% RSLogix 500 project PROJECT10.RSS, saved by version 8.30.00.16 %
PROJECT "PROJ_9"    % processor: Bul.1763 MicroLogix 1100 Series B %

PROGRAM FILES
  LAD 2 "MAIN"  5 rungs
  LAD 3 "I/O"  11 rungs
  LAD 4 "CONTROL"  6 rungs
  LAD 5 "ALARMS"  5 rungs

DATA FILES
  O0 OUTPUT  5 elements
  I1 INPUT  7 elements
  S2 STATUS  66 elements
  B3 BINARY  2 elements
  T4 TIMER  4 elements
  C5 COUNTER  1 elements
  R6 CONTROL  1 elements
  N7 INTEGER  2 elements
  F8 FLOAT  1 elements

LADDER 2 "MAIN"
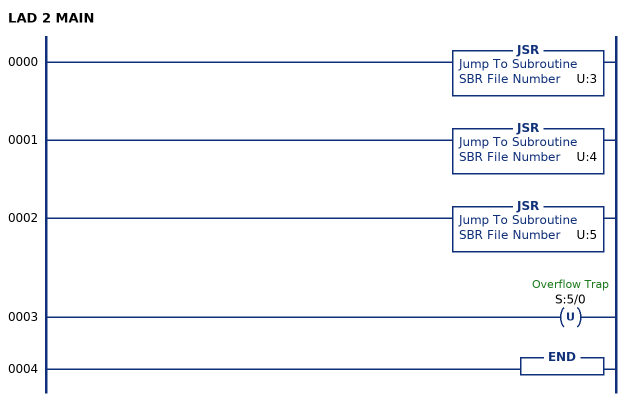
% Rung: 0 %
SOR JSR U:3 EOR
% Rung: 1 %
SOR JSR U:4 EOR
% Rung: 2 %
SOR JSR U:5 EOR
% Rung: 3 %
SOR OTU S:5/0 EOR
%   S:5/0  "Overflow Trap" %
% Rung: 4 %
SOR END EOR

LADDER 3 "I/O"
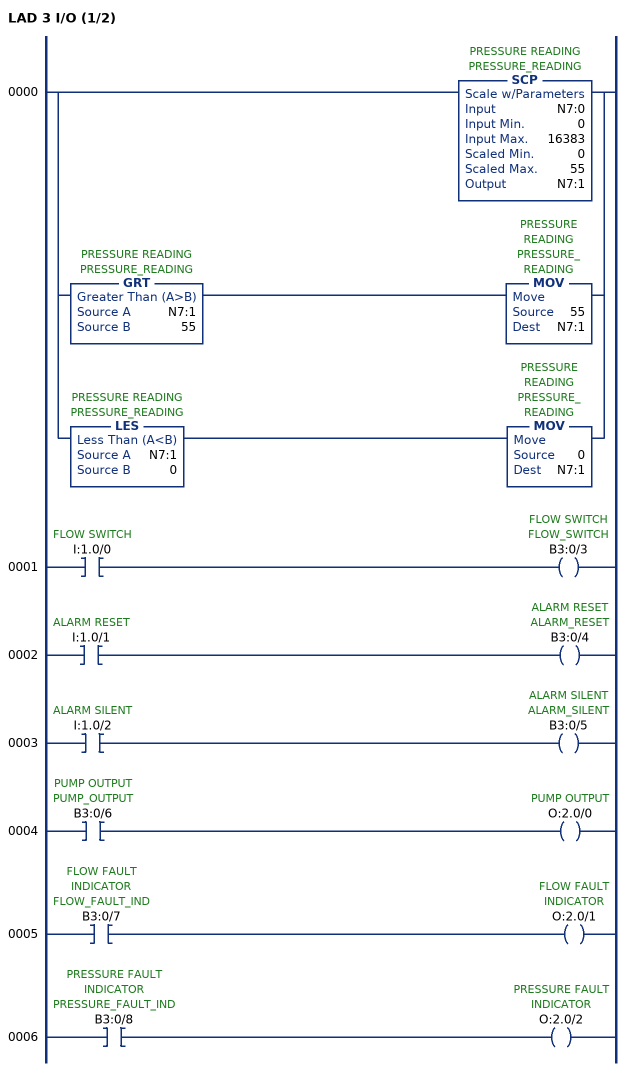
% Rung: 0 %
SOR BST SCP N7:0 0 16383 0 55 N7:1 NXB GRT N7:1 55 MOV 55 N7:1 NXB LES N7:1 0 MOV 0 N7:1 BND EOR
%   N7:0  "PRESSURE INPUT" %
%   N7:1  PRESSURE_READING  "PRESSURE READING" %
% Rung: 1 %
SOR XIC I:1.0/0 OTE B3:0/3 EOR
%   I:1.0/0  "FLOW SWITCH" %
%   B3:0/3  FLOW_SWITCH  "FLOW SWITCH" %
% Rung: 2 %
SOR XIC I:1.0/1 OTE B3:0/4 EOR
%   I:1.0/1  "ALARM RESET" %
%   B3:0/4  ALARM_RESET  "ALARM RESET" %
% Rung: 3 %
SOR XIC I:1.0/2 OTE B3:0/5 EOR
%   I:1.0/2  "ALARM SILENT" %
%   B3:0/5  ALARM_SILENT  "ALARM SILENT" %
% Rung: 4 %
SOR XIC B3:0/6 OTE O:2.0/0 EOR
%   B3:0/6  PUMP_OUTPUT  "PUMP OUTPUT" %
%   O:2.0/0  "PUMP OUTPUT" %
% Rung: 5 %
SOR XIC B3:0/7 OTE O:2.0/1 EOR
%   B3:0/7  FLOW_FAULT_IND  "FLOW FAULT INDICATOR" %
%   O:2.0/1  "FLOW FAULT INDICATOR" %
% Rung: 6 %
SOR XIC B3:0/8 OTE O:2.0/2 EOR
%   B3:0/8  PRESSURE_FAULT_IND  "PRESSURE FAULT INDICATOR" %
%   O:2.0/2  "PRESSURE FAULT INDICATOR" %

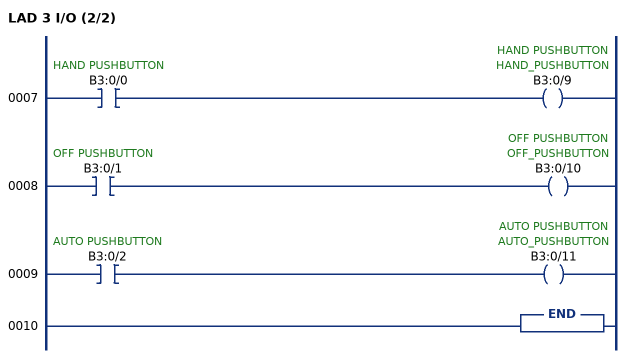
% Rung: 7 %
SOR XIC B3:0/0 OTE B3:0/9 EOR
%   B3:0/0  "HAND PUSHBUTTON" %
%   B3:0/9  HAND_PUSHBUTTON  "HAND PUSHBUTTON" %
% Rung: 8 %
SOR XIC B3:0/1 OTE B3:0/10 EOR
%   B3:0/1  "OFF PUSHBUTTON" %
%   B3:0/10  OFF_PUSHBUTTON  "OFF PUSHBUTTON" %
% Rung: 9 %
SOR XIC B3:0/2 OTE B3:0/11 EOR
%   B3:0/2  "AUTO PUSHBUTTON" %
%   B3:0/11  AUTO_PUSHBUTTON  "AUTO PUSHBUTTON" %
% Rung: 10 %
SOR END EOR

LADDER 4 "CONTROL"
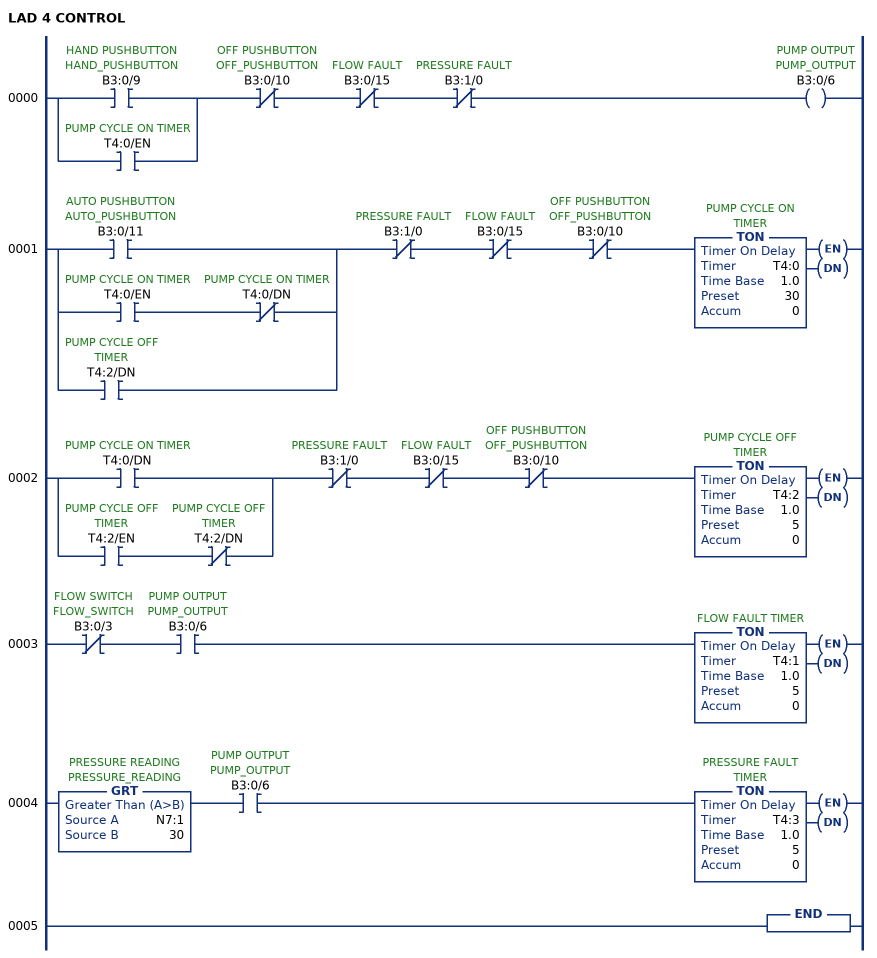
% Rung: 0 %
SOR BST XIC B3:0/9 NXB XIC T4:0/EN BND XIO B3:0/10 XIO B3:0/15 XIO B3:1/0 OTE B3:0/6 EOR
%   B3:0/9  HAND_PUSHBUTTON  "HAND PUSHBUTTON" %
%   T4:0  "PUMP CYCLE ON TIMER" %
%   B3:0/10  OFF_PUSHBUTTON  "OFF PUSHBUTTON" %
%   B3:0/15  "FLOW FAULT" %
%   B3:1/0  "PRESSURE FAULT" %
%   B3:0/6  PUMP_OUTPUT  "PUMP OUTPUT" %
% Rung: 1 %
SOR BST XIC B3:0/11 NXB XIC T4:0/EN XIO T4:0/DN NXB XIC T4:2/DN BND XIO B3:1/0 XIO B3:0/15 XIO B3:0/10 TON T4:0 1.0 30 0 EOR
%   B3:0/11  AUTO_PUSHBUTTON  "AUTO PUSHBUTTON" %
%   T4:0  "PUMP CYCLE ON TIMER" %
%   T4:2  "PUMP CYCLE OFF TIMER" %
%   B3:1/0  "PRESSURE FAULT" %
%   B3:0/15  "FLOW FAULT" %
%   B3:0/10  OFF_PUSHBUTTON  "OFF PUSHBUTTON" %
% Rung: 2 %
SOR BST XIC T4:0/DN NXB XIC T4:2/EN XIO T4:2/DN BND XIO B3:1/0 XIO B3:0/15 XIO B3:0/10 TON T4:2 1.0 5 0 EOR
%   T4:0  "PUMP CYCLE ON TIMER" %
%   T4:2  "PUMP CYCLE OFF TIMER" %
%   B3:1/0  "PRESSURE FAULT" %
%   B3:0/15  "FLOW FAULT" %
%   B3:0/10  OFF_PUSHBUTTON  "OFF PUSHBUTTON" %
% Rung: 3 %
SOR XIO B3:0/3 XIC B3:0/6 TON T4:1 1.0 5 0 EOR
%   B3:0/3  FLOW_SWITCH  "FLOW SWITCH" %
%   B3:0/6  PUMP_OUTPUT  "PUMP OUTPUT" %
%   T4:1  "FLOW FAULT TIMER" %
% Rung: 4 %
SOR GRT N7:1 30 XIC B3:0/6 TON T4:3 1.0 5 0 EOR
%   N7:1  PRESSURE_READING  "PRESSURE READING" %
%   B3:0/6  PUMP_OUTPUT  "PUMP OUTPUT" %
%   T4:3  "PRESSURE FAULT TIMER" %
% Rung: 5 %
SOR END EOR

LADDER 5 "ALARMS"
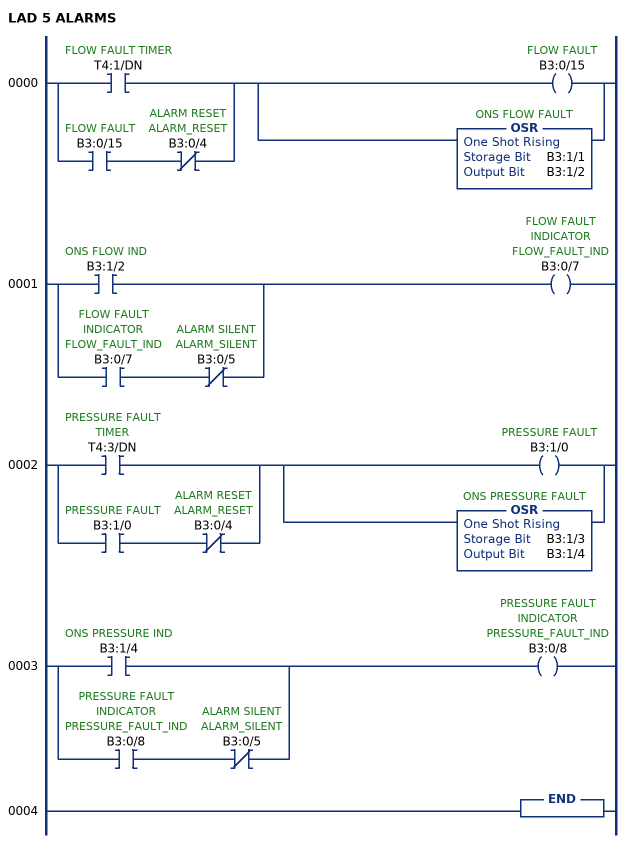
% Rung: 0 %
SOR BST XIC T4:1/DN NXB XIC B3:0/15 XIO B3:0/4 BND BST OTE B3:0/15 NXB OSR B3:1/1 B3:1/2 BND EOR
%   T4:1  "FLOW FAULT TIMER" %
%   B3:0/15  "FLOW FAULT" %
%   B3:0/4  ALARM_RESET  "ALARM RESET" %
%   B3:1/1  "ONS FLOW FAULT" %
%   B3:1/2  "ONS FLOW IND" %
% Rung: 1 %
SOR BST XIC B3:1/2 NXB XIC B3:0/7 XIO B3:0/5 BND OTE B3:0/7 EOR
%   B3:1/2  "ONS FLOW IND" %
%   B3:0/7  FLOW_FAULT_IND  "FLOW FAULT INDICATOR" %
%   B3:0/5  ALARM_SILENT  "ALARM SILENT" %
% Rung: 2 %
SOR BST XIC T4:3/DN NXB XIC B3:1/0 XIO B3:0/4 BND BST OTE B3:1/0 NXB OSR B3:1/3 B3:1/4 BND EOR
%   T4:3  "PRESSURE FAULT TIMER" %
%   B3:1/0  "PRESSURE FAULT" %
%   B3:0/4  ALARM_RESET  "ALARM RESET" %
%   B3:1/3  "ONS PRESSURE FAULT" %
%   B3:1/4  "ONS PRESSURE IND" %
% Rung: 3 %
SOR BST XIC B3:1/4 NXB XIC B3:0/8 XIO B3:0/5 BND OTE B3:0/8 EOR
%   B3:1/4  "ONS PRESSURE IND" %
%   B3:0/8  PRESSURE_FAULT_IND  "PRESSURE FAULT INDICATOR" %
%   B3:0/5  ALARM_SILENT  "ALARM SILENT" %
% Rung: 4 %
SOR END EOR

OTHER DOCUMENTED ADDRESSES
  B3:0/12  "ONS FLOW FAULT"
  B3:0/13  "PUMP CYCLE"
  B3:0/14  "AUTO MODE"

DATA TABLE (non-zero values as saved)
DATA T4
% .PRE .ACC %
% T4:0 % 30 0
% T4:1 % 5 0
% T4:2 % 5 0
% T4:3 % 5 0
